PROGRAM ChargeTime
VAR

	lca_charge_cal	 : ARRAY [1..8] OF LCA_CAL;
	i				 : INT := 1; // 1-8 instances
	j				 : INT := 1; //1 - 8 ch
	m				 : INT := 1;
	
	a				 : INT := 1; 
	
	Q				 : REAL := 1; // Charge
	Current			 : REAL := 0.1; //100mA
	
	longestChargeTime: REAL;
	
END_VAR

(*IF HMI_DB.RemoteModeSelected = FALSE THEN 
	HMI_DB.TDKLoad[1].PSratedV := 12; //veto at 10
	HMI_DB.TDKLoad[2].PSratedV := 12;
	HMI_DB.TDKLoad[3].PSratedV := 12;
	HMI_DB.TDKLoad[4].PSratedV := 12;
	HMI_DB.TDKLoad[5].PSratedV := 12;
	HMI_DB.TDKLoad[6].PSratedV := 12;
	HMI_DB.TDKLoad[7].PSratedV := 50; //veto at 35
	HMI_DB.TDKLoad[8].PSratedV := 50;
	HMI_DB.GLSLoad.PSratedV := 30;
	
	HMI_DB.TDKLoad[1].TotalCapacitance := 10000;
	HMI_DB.TDKLoad[2].TotalCapacitance := 10000;
	HMI_DB.TDKLoad[3].TotalCapacitance := 10000;
	HMI_DB.TDKLoad[4].TotalCapacitance := 16000;
	HMI_DB.TDKLoad[5].TotalCapacitance := 16000;
	HMI_DB.TDKLoad[6].TotalCapacitance := 16000;
	HMI_DB.TDKLoad[7].TotalCapacitance := 1200;
	HMI_DB.TDKLoad[8].TotalCapacitance := 1200;
	HMI_DB.GLSLoad.TotalCapacitance := 200;
	
END_IF*)

//veto
//this should not happen
FOR m := 1 TO 6 BY 1 DO
	IF Setpoints.TDKLoad[m].RequiredChargedV <= -2 THEN
		Setpoints.TDKLoad[m].RequiredChargedV := -2;
	END_IF	
END_FOR

IF Setpoints.GLSLoad.RequiredChargedV <= 0 THEN
	Setpoints.GLSLoad.RequiredChargedV := 0;
END_IF	

//ch 1 - 3
IF Setpoints.TDKLoad[1].RequiredChargedV >= 10 THEN
	Setpoints.TDKLoad[1].RequiredChargedV := 10;
	ELSIF Setpoints.TDKLoad[1].RequiredChargedV < 0 THEN
		Setpoints.TDKLoad[1].RequiredChargedV := ABS(Setpoints.TDKLoad[1].RequiredChargedV); 
END_IF
IF Setpoints.TDKLoad[2].RequiredChargedV >= 10 THEN
	Setpoints.TDKLoad[2].RequiredChargedV := 10;
	ELSIF Setpoints.TDKLoad[2].RequiredChargedV < 0 THEN
		Setpoints.TDKLoad[2].RequiredChargedV := ABS(Setpoints.TDKLoad[2].RequiredChargedV); 	
END_IF
IF Setpoints.TDKLoad[3].RequiredChargedV >= 10 THEN
	Setpoints.TDKLoad[3].RequiredChargedV := 10;
	ELSIF Setpoints.TDKLoad[3].RequiredChargedV < 0 THEN
		Setpoints.TDKLoad[3].RequiredChargedV := ABS(Setpoints.TDKLoad[3].RequiredChargedV); 	
END_IF
//ch 4-6
IF Setpoints.TDKLoad[4].RequiredChargedV >= 12 THEN
	Setpoints.TDKLoad[4].RequiredChargedV := 12;
	ELSIF Setpoints.TDKLoad[4].RequiredChargedV < 0 THEN
		Setpoints.TDKLoad[4].RequiredChargedV := ABS(Setpoints.TDKLoad[4].RequiredChargedV); 	
END_IF
IF Setpoints.TDKLoad[5].RequiredChargedV >= 12 THEN
	Setpoints.TDKLoad[5].RequiredChargedV := 12;
	ELSIF Setpoints.TDKLoad[5].RequiredChargedV < 0 THEN
		Setpoints.TDKLoad[5].RequiredChargedV := ABS(Setpoints.TDKLoad[5].RequiredChargedV); 	
END_IF
IF Setpoints.TDKLoad[6].RequiredChargedV >= 12 THEN
	Setpoints.TDKLoad[6].RequiredChargedV := 12;
	ELSIF Setpoints.TDKLoad[6].RequiredChargedV < 0 THEN
		Setpoints.TDKLoad[6].RequiredChargedV := ABS(Setpoints.TDKLoad[6].RequiredChargedV); 	
END_IF
//ch 7 - 8
IF Setpoints.TDKLoad[7].RequiredChargedV >= 35 THEN
	Setpoints.TDKLoad[7].RequiredChargedV := 35;
	ELSIF Setpoints.TDKLoad[7].RequiredChargedV <= 0  THEN
		Setpoints.TDKLoad[7].RequiredChargedV := 0; 	
END_IF
IF Setpoints.TDKLoad[8].RequiredChargedV >= 35 THEN
	Setpoints.TDKLoad[8].RequiredChargedV := 35;
	ELSIF Setpoints.TDKLoad[8].RequiredChargedV <= 0 THEN
		Setpoints.TDKLoad[8].RequiredChargedV := ABS(Setpoints.TDKLoad[8].RequiredChargedV); 	
END_IF
IF Setpoints.GLSLoad.RequiredChargedV >= 30 THEN
	Setpoints.GLSLoad.RequiredChargedV := 30;
	ELSIF Setpoints.GLSLoad.RequiredChargedV <= 0 THEN
		Setpoints.GLSLoad.RequiredChargedV := 0; 	
END_IF

//mapping hmi input to setpoints
FOR j := 1 TO 8 BY 1 DO	
	Setpoints.TDKLoad[j].TotalCapacitance	:= HMI_DB.TDKLoad[j].TotalCapacitance;
	Setpoints.TDKLoad[j].PSratedV 			:= HMI_DB.TDKLoad[j].PSratedV;
	//Setpoints.PeakBank[m].RequiredChargedV	:= Recipe.PeakBank[m].RequiredChargedV; //only thing that comes from the main plc recipe
	Setpoints.TDKLoad[j].wLCA				:= HMI_DB.TDKLoad[j].wLCA;
	Setpoints.TDKLoad[j].NumOfCharger		:= HMI_DB.TDKLoad[j].NumOfCharger;	
	
	Setpoints.TDKLoad[j].TotalCapacitance	:= HMI_DB.TDKLoad[j].TotalCapacitance;
	Setpoints.TDKLoad[j].PSratedV 			:= HMI_DB.TDKLoad[j].PSratedV;
	//Setpoints.SustBank[m].RequiredChargedV	:= Recipe.SustBank[m].RequiredChargedV; //only thing that comes from the main plc recipe
	Setpoints.TDKLoad[j].wLCA				:= HMI_DB.TDKLoad[j].wLCA;
	Setpoints.TDKLoad[j].NumOfCharger		:= HMI_DB.TDKLoad[j].NumOfCharger;	
	//charge time delay and elapse for HMI
	ChargeTime_DB.ChargeTimeStartDelay[j] := TIME_TO_INT((ChargeTime_DB.ChargerDelay_PT[j] - ChargeTime_DB.ChargerDelay_ET[j])/1000);
	ChargeTime_DB.ChargingTimeElapse[j] := TIME_TO_INT((ChargeTime_DB.ChargingTimeElapse_TON[j].PT - ChargeTime_DB.ChargingTimeElapse_TON[j].ET)/1000);
END_FOR

ChargeTime_DB.PreFormChargeTimeStartDelay := TIME_TO_INT((ChargeTime_DB.PreFormChargeTime_PT - ChargeTime_DB.PreFormChargeTime_ET)/1000);
ChargeTime_DB.PreFormChargingTimeElapse := TIME_TO_INT((ChargeTime_DB.PreFormChargingTimeElapse_TON.PT - ChargeTime_DB.PreFormChargingTimeElapse_TON.ET)/1000);

//GLS 3
Setpoints.GLSLoad.TotalCapacitance	:= HMI_DB.GLSLoad.TotalCapacitance;
Setpoints.GLSLoad.PSratedV 			:= HMI_DB.GLSLoad.PSratedV;
//Setpoints.PreFormBank.RequiredChargedV	:= Recipe.PreFormBank.RequiredChargedV; //only thing that comes from the main plc recipe
//Setpoints.GLSLoad.wLCA				:= HMI_DB.GLSLoad.wLCA;
Setpoints.GLSLoad.NumOfCharger		:= HMI_DB.GLSLoad.NumOfCharger;	

//chg time
FOR i := 1 TO 8 BY 1 DO
	lca_charge_cal[i](	PSratedV := Setpoints.TDKLoad[i].PSratedV, 
						RequiredChargeV := Setpoints.TDKLoad[i].RequiredChargedV, 
						LoadCapacitance := Setpoints.TDKLoad[i].TotalCapacitance, 
						NumOfCharger := Setpoints.TDKLoad[i].NumOfCharger, 
						wLCA := Setpoints.TDKLoad[i].wLCA
						);

	MCP_IO.Charger[i].ChargeTime.timeToChargeLoad := lca_charge_cal[i].TimeToChargeLoad;
	MCP_IO.Charger[i].ChargeTime.Power := lca_charge_cal[i].RespectedPower;
END_FOR


//gls - gls3 is preform cap charger
Q := 1000* Setpoints.GLSLoad.RequiredChargedV * (Setpoints.GLSLoad.TotalCapacitance / 1000000);
MCP_IO.GLS3_Load.timeToChargeLoad := Q / Current;
MCP_IO.GLS3_Load.Power := 1000*Setpoints.GLSLoad.RequiredChargedV * Current;

//find the longest charge time.  //need more work
longestChargeTime := MAX( MCP_IO.Charger[1].ChargeTime.timeToChargeLoad,
							MCP_IO.Charger[2].ChargeTime.timeToChargeLoad,
							MCP_IO.Charger[3].ChargeTime.timeToChargeLoad,
							MCP_IO.Charger[4].ChargeTime.timeToChargeLoad,
							MCP_IO.Charger[5].ChargeTime.timeToChargeLoad,
							MCP_IO.Charger[6].ChargeTime.timeToChargeLoad,
							MCP_IO.Charger[7].ChargeTime.timeToChargeLoad,
							MCP_IO.Charger[8].ChargeTime.timeToChargeLoad, 
							MCP_IO.GLS3_Load.timeToChargeLoad);

ChargeTime_DB.LongestChargeTime_PT := REAL_TO_TIME (1000*longestChargeTime);

FOR a := 1 TO 8 BY 1 DO
	IF (longestChargeTime - MCP_IO.Charger[a].ChargeTime.timeToChargeLoad) >= 0 THEN
		ChargeTime_DB.ChargerDelay_PT[a] := REAL_TO_TIME (1000*(longestChargeTime - MCP_IO.Charger[a].ChargeTime.timeToChargeLoad));
		ELSE 
			ChargeTime_DB.ChargerDelay_PT[a] := REAL_TO_TIME (1000*(MCP_IO.Charger[a].ChargeTime.timeToChargeLoad - longestChargeTime));
	END_IF;		
		
	//IF (longestChargeTime - MCP_IO.Charger[a+3].ChargeTime.timeToChargeLoad) >= 0 THEN
	//	ChargeTime_DB.SustChargeTime_PT[a] := REAL_TO_TIME (1000*(longestChargeTime - MCP_IO.Charger[a+3].ChargeTime.timeToChargeLoad));	
	//END_IF;	
	
END_FOR;


(*IF (longestChargeTime - MCP_IO.Charger[7].ChargeTime.timeToChargeLoad) >= 0 THEN
	ChargeTime_DB.FormChargeTime_PT[1] := REAL_TO_TIME (1000*(longestChargeTime - MCP_IO.Charger[7].ChargeTime.timeToChargeLoad));	
END_IF;	
IF (longestChargeTime - MCP_IO.Charger[8].ChargeTime.timeToChargeLoad) >= 0 THEN
	ChargeTime_DB.FormChargeTime_PT[2] := REAL_TO_TIME (1000*(longestChargeTime - MCP_IO.Charger[8].ChargeTime.timeToChargeLoad));	
END_IF;	
*)
IF (longestChargeTime - MCP_IO.GLS3_Load.timeToChargeLoad) >= 0 THEN
		ChargeTime_DB.PreFormChargeTime_PT := REAL_TO_TIME (1000*(longestChargeTime - MCP_IO.GLS3_Load.timeToChargeLoad));
		ELSE
			ChargeTime_DB.PreFormChargeTime_PT := REAL_TO_TIME (1000*(MCP_IO.GLS3_Load.timeToChargeLoad -longestChargeTime));
END_IF;



IF i > 8 THEN 
	i := 0;
END_IF

IF j > 8 THEN
	j := 0;
END_IF

IF m > 6 THEN
	m := 0;
END_IF

IF a > 8 THEN 
	a := 1;
END_IF;

END_PROGRAM

(* stored: Version 1.1.0.1, ProductVersion 3.1.4024.11
   POU ChargeTime: Id {28824270-3930-44b7-bfe2-d4b07042cd6b}, SpecialFunc None *)
